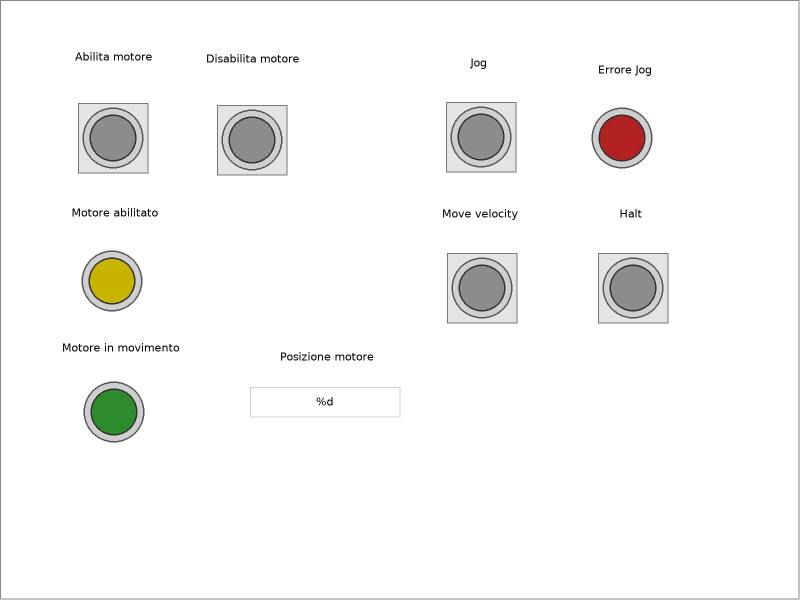
VISUALIZATION Visualization  // 800x600
    Label (39,42 150x30), "Abilita motore"
    PushSwitch (78,103 70x70), variable: GVL.pBEnableMotor, behaviour: TAP, style: Switch-PushSwitch-Gray
    Lamp1 (77,246 70x70), variable: GVL.motorIsReallyEnabled, style: Lamp-Lamp1-Yellow
    Label (40,198 150x30), "Motore abilitato"
    Label (178,44 150x30), "Disabilita motore"
    PushSwitch (217,105 70x70), variable: GVL.pbDisableMotor, behaviour: TAP, style: Switch-PushSwitch-Gray
    PushSwitch (446,102 70x70), variable: GVL.pBJog, behaviour: TAP, style: Switch-PushSwitch-Gray
    Label (404,48 150x30), "Jog"
    Lamp1 (587,103 70x70), variable: GVL.jogError, style: Lamp-Lamp1-Red
    Label (550,55 150x30), "Errore Jog"
    Lamp1 (79,377 70x70), variable: GVL.axis.Status.Moving, style: Lamp-Lamp1-Green
    Label (46,333 150x30), "Motore in movimento"
    Textfield (250,387 150x30), "%d", text variable: GVL.axis.NcToPlc.ActPos
    Label (252,342 150x30), "Posizione motore"
    Label (405,199 150x30), "Move velocity"
    PushSwitch (447,253 70x70), variable: GVL.pBMoveVelocity, behaviour: TAP, style: Switch-PushSwitch-Gray
    Label (556,199 150x30), "Halt"
    PushSwitch (598,253 70x70), variable: GVL.pBHalt, behaviour: TAP, style: Switch-PushSwitch-Gray
END_VISUALIZATION

(* stored: Version 1.1.0.1, ProductVersion 3.1.4024.12
   Visu Visualization: Id {40c7f54e-cf99-43a0-96ab-a2c16cccd96c} *)
